// TIA Portal V15.1 export
// export: Created 2024-05-17T05:38:39.7334775Z, ExportSetting WithDefaults, DisplayName Totally Integrated Automation Portal, DisplayVersion V15.1 Update 5, DisplayName TIA Portal Openness, DisplayVersion V15.1 Update 5, DisplayName SINAMICS Startdrive Advanced, DisplayVersion V15.1, DisplayName G130, G150, S120, S150, SINAMICS MV, S210, DisplayVersion V15.1, DisplayName G110M, G120, G120C, G120D, G120P, DisplayVersion V15.1, DisplayName STEP 7 Professional, DisplayVersion V15.1 Update 5, DisplayName STEP 7 Safety, DisplayVersion V15.1, DisplayName WinCC Professional, DisplayVersion V15.1 Update 5, DisplayName SIMATIC Visualization Architect, DisplayVersion V15.1
FUNCTION_BLOCK "LGBJoyStick"   // FB6647, FBD
TITLE = LGBJoyStick
{ S7_Optimized_Access := 'TRUE' }
AUTHOR : VCC
FAMILY : Tooling
VERSION : 0.1
// ============================================================================
// This module works as a (virtual) joystick.
// The module can be used to force/block orders in a specific direction (lifts, cross conveyors, ...)
// ============================================================================
// stored: AutoNumber false, IsIECCheckEnabled true, IsRetainMemResEnabled false, MemoryReserve 100, SetENOAutomatically False, UDAEnableTagReadback false
   VAR_INPUT
      I_ExtBtnUp { ExternalAccessible := 'False'; ExternalVisible := 'False'; ExternalWritable := 'False'} : Bool;   // External Button Up
      I_ExtBtnRight { ExternalAccessible := 'False'; ExternalVisible := 'False'; ExternalWritable := 'False'} : Bool;   // External Button Right
      I_ExtBtnDown { ExternalAccessible := 'False'; ExternalVisible := 'False'; ExternalWritable := 'False'} : Bool;   // External Button Down
      I_ExtBtnLeft { ExternalAccessible := 'False'; ExternalVisible := 'False'; ExternalWritable := 'False'} : Bool;   // External Button Left
      I_OutOfUse { ExternalAccessible := 'False'; ExternalVisible := 'False'; ExternalWritable := 'False'} : Bool;   // Object out of use / Out of use
   END_VAR
   VAR_OUTPUT
      O_BtnMiddle { ExternalAccessible := 'False'; ExternalVisible := 'False'; ExternalWritable := 'False'} : Bool;   // Btn Middle Active
      O_BtnUp { ExternalAccessible := 'False'; ExternalVisible := 'False'; ExternalWritable := 'False'} : Bool;   // Btn Up Active
      O_BtnRight { ExternalAccessible := 'False'; ExternalVisible := 'False'; ExternalWritable := 'False'} : Bool;   // Btn Right Active
      O_BtnDown { ExternalAccessible := 'False'; ExternalVisible := 'False'; ExternalWritable := 'False'} : Bool;   // Btn Down Active
      O_BtnLeft { ExternalAccessible := 'False'; ExternalVisible := 'False'; ExternalWritable := 'False'} : Bool;   // Btn Left Active
      O_AnyBtnActive { ExternalAccessible := 'False'; ExternalVisible := 'False'; ExternalWritable := 'False'} : Bool;   // Any Button Active
      O_AlarmABCondition { ExternalAccessible := 'False'; ExternalVisible := 'False'; ExternalWritable := 'False'} : Bool;   // Alarm AB Condition
      O_AlarmA { ExternalAccessible := 'False'; ExternalVisible := 'False'; ExternalWritable := 'False'} : Bool;   // Alarm A
      O_AlarmB { ExternalAccessible := 'False'; ExternalVisible := 'False'; ExternalWritable := 'False'} : Bool;   // Alarm B
      O_AlarmC { ExternalAccessible := 'False'; ExternalVisible := 'False'; ExternalWritable := 'False'} : Bool;   // Alarm C
      O_AlarmD { ExternalAccessible := 'False'; ExternalVisible := 'False'; ExternalWritable := 'False'} : Bool;   // Alarm D
      H_AlarmDWord { ExternalAccessible := 'False'; ExternalVisible := 'False'; ExternalWritable := 'False'} : DWord;   // Alarm Word
   END_VAR
   VAR_IN_OUT
      H_HMI : "H_HMI";   // Icon Animation
      H_GBJoyStick : "H_GBJoyStick";   // Animation
      C_GBJoyStickConfig : "JoyStickConfig";   // Config
   END_VAR
   VAR
      AD_BtnMiddleActByHMI { ExternalAccessible := 'False'; ExternalVisible := 'False'; ExternalWritable := 'False'} : Bool;   // JoyStick - Button Middle is Active by HMI
      AD_BtnUpActByHMI { ExternalAccessible := 'False'; ExternalVisible := 'False'; ExternalWritable := 'False'} : Bool;   // JoyStick - Button Up is Active by HMI
      AD_BtnRightActByHMI { ExternalAccessible := 'False'; ExternalVisible := 'False'; ExternalWritable := 'False'} : Bool;   // JoyStick - Button Right is Active by HMI
      AD_BtnDownActByHMI { ExternalAccessible := 'False'; ExternalVisible := 'False'; ExternalWritable := 'False'} : Bool;   // JoyStick - Button Down is Active by HMI
      AD_BtnLeftActByHMI { ExternalAccessible := 'False'; ExternalVisible := 'False'; ExternalWritable := 'False'} : Bool;   // JoyStick - Button Left is Active by HMI
      AD_BtnUpActByExtCmd { ExternalAccessible := 'False'; ExternalVisible := 'False'; ExternalWritable := 'False'} : Bool;   // JoyStick - Button Up is Active by External command
      AD_BtnRightActByExtCmd { ExternalAccessible := 'False'; ExternalVisible := 'False'; ExternalWritable := 'False'} : Bool;   // JoyStick - Button Right is Active by External command
      AD_BtnDownActByExtCmd { ExternalAccessible := 'False'; ExternalVisible := 'False'; ExternalWritable := 'False'} : Bool;   // JoyStick - Button Down is Active by External command
      AD_BtnLeftActByExtCmd { ExternalAccessible := 'False'; ExternalVisible := 'False'; ExternalWritable := 'False'} : Bool;   // JoyStick - Button Left is Active by External command
      BtnHMICmd { ExternalAccessible := 'False'; ExternalVisible := 'False'; ExternalWritable := 'False'} : Struct   // HMI Commands
         BtnMiddle { ExternalAccessible := 'False'; ExternalVisible := 'False'; ExternalWritable := 'False'} : Bool;   // Btn Middle Selected
         BtnUp { ExternalAccessible := 'False'; ExternalVisible := 'False'; ExternalWritable := 'False'} : Bool;   // Btn Up Selected
         BtnRight { ExternalAccessible := 'False'; ExternalVisible := 'False'; ExternalWritable := 'False'} : Bool;   // Btn Right Selected
         BtnDown { ExternalAccessible := 'False'; ExternalVisible := 'False'; ExternalWritable := 'False'} : Bool;   // Btn Down Selected
         BtnLeft { ExternalAccessible := 'False'; ExternalVisible := 'False'; ExternalWritable := 'False'} : Bool;   // Btn Left Selected
      END_STRUCT;
      BtnResult { ExternalAccessible := 'False'; ExternalVisible := 'False'; ExternalWritable := 'False'} : Struct   // Buttons
         BtnMiddle { ExternalAccessible := 'False'; ExternalVisible := 'False'; ExternalWritable := 'False'} : Bool;   // Btn Middle Selected
         BtnUp { ExternalAccessible := 'False'; ExternalVisible := 'False'; ExternalWritable := 'False'} : Bool;   // Btn Up Selected
         BtnRight { ExternalAccessible := 'False'; ExternalVisible := 'False'; ExternalWritable := 'False'} : Bool;   // Btn Right Selected
         BtnDown { ExternalAccessible := 'False'; ExternalVisible := 'False'; ExternalWritable := 'False'} : Bool;   // Btn Down Selected
         BtnLeft { ExternalAccessible := 'False'; ExternalVisible := 'False'; ExternalWritable := 'False'} : Bool;   // Btn Left Selected
      END_STRUCT;
      Cmd { ExternalAccessible := 'False'; ExternalVisible := 'False'; ExternalWritable := 'False'} : Struct   // Commands
         Middle { ExternalAccessible := 'False'; ExternalVisible := 'False'; ExternalWritable := 'False'} : Bool;   // Middle Command
         BlockUp { ExternalAccessible := 'False'; ExternalVisible := 'False'; ExternalWritable := 'False'} : Bool;   // Block Up Command
         BlockRight { ExternalAccessible := 'False'; ExternalVisible := 'False'; ExternalWritable := 'False'} : Bool;   // Block Right Command
         BlockDown { ExternalAccessible := 'False'; ExternalVisible := 'False'; ExternalWritable := 'False'} : Bool;   // Block Down Command
         BlockLeft { ExternalAccessible := 'False'; ExternalVisible := 'False'; ExternalWritable := 'False'} : Bool;   // Block Left Command
         ForceUp { ExternalAccessible := 'False'; ExternalVisible := 'False'; ExternalWritable := 'False'} : Bool;   // Force Up Command
         ForceRight { ExternalAccessible := 'False'; ExternalVisible := 'False'; ExternalWritable := 'False'} : Bool;   // Force Right Command
         ForceDown { ExternalAccessible := 'False'; ExternalVisible := 'False'; ExternalWritable := 'False'} : Bool;   // Force Down Command
         ForceLeft { ExternalAccessible := 'False'; ExternalVisible := 'False'; ExternalWritable := 'False'} : Bool;   // Force Left Command
      END_STRUCT;
      Anim { ExternalAccessible := 'False'; ExternalVisible := 'False'; ExternalWritable := 'False'} : Struct   // HMI Animation
         HoldMiddleOff { ExternalAccessible := 'False'; ExternalVisible := 'False'; ExternalWritable := 'False'} : Bool;   // Anim Hold Middle Button Off
         HoldMiddleOn { ExternalAccessible := 'False'; ExternalVisible := 'False'; ExternalWritable := 'False'} : Bool;   // Anim Hold Middle Button On
         ForceUpOff { ExternalAccessible := 'False'; ExternalVisible := 'False'; ExternalWritable := 'False'} : Bool;   // Anim Force Up Button Off
         ForceUpOn { ExternalAccessible := 'False'; ExternalVisible := 'False'; ExternalWritable := 'False'} : Bool;   // Anim Force Up Button On
         BlockUpOff { ExternalAccessible := 'False'; ExternalVisible := 'False'; ExternalWritable := 'False'} : Bool;   // Anim Block Up Button Off
         BlockUpOn { ExternalAccessible := 'False'; ExternalVisible := 'False'; ExternalWritable := 'False'} : Bool;   // Anim Block Up Button On
         ForceRightOff { ExternalAccessible := 'False'; ExternalVisible := 'False'; ExternalWritable := 'False'} : Bool;   // Anim Force Right Button Off
         ForceRightOn { ExternalAccessible := 'False'; ExternalVisible := 'False'; ExternalWritable := 'False'} : Bool;   // Anim Force Right Button On
         BlockRightOff { ExternalAccessible := 'False'; ExternalVisible := 'False'; ExternalWritable := 'False'} : Bool;   // Anim Block Right Button Off
         BlockRightOn { ExternalAccessible := 'False'; ExternalVisible := 'False'; ExternalWritable := 'False'} : Bool;   // Anim Block Right Button On
         ForceDownOff { ExternalAccessible := 'False'; ExternalVisible := 'False'; ExternalWritable := 'False'} : Bool;   // Anim Force Down Button Off
         ForceDownOn { ExternalAccessible := 'False'; ExternalVisible := 'False'; ExternalWritable := 'False'} : Bool;   // Anim Force Down Button On
         BlockDownOff { ExternalAccessible := 'False'; ExternalVisible := 'False'; ExternalWritable := 'False'} : Bool;   // Anim Block Down Button Off
         BlockDownOn { ExternalAccessible := 'False'; ExternalVisible := 'False'; ExternalWritable := 'False'} : Bool;   // Anim Block Down Button On
         ForceLeftOff { ExternalAccessible := 'False'; ExternalVisible := 'False'; ExternalWritable := 'False'} : Bool;   // Anim Force Left Button Off
         ForceLeftOn { ExternalAccessible := 'False'; ExternalVisible := 'False'; ExternalWritable := 'False'} : Bool;   // Anim Force Left Button On
         BlockLeftOff { ExternalAccessible := 'False'; ExternalVisible := 'False'; ExternalWritable := 'False'} : Bool;   // Anim Block Left Button Off
         BlockLeftOn { ExternalAccessible := 'False'; ExternalVisible := 'False'; ExternalWritable := 'False'} : Bool;   // Anim Block Left Button On
      END_STRUCT;
      ExtBtnActive { ExternalAccessible := 'False'; ExternalVisible := 'False'; ExternalWritable := 'False'} : Bool;   // External Button Active
   END_VAR
   VAR RETAIN
      BtnMiddleAct { ExternalAccessible := 'False'; ExternalVisible := 'False'; ExternalWritable := 'False'} : Bool;   // Btn Middle Active memory
      BtnUpAct { ExternalAccessible := 'False'; ExternalVisible := 'False'; ExternalWritable := 'False'} : Bool;   // Btn Up Active memory
      BtnRightAct { ExternalAccessible := 'False'; ExternalVisible := 'False'; ExternalWritable := 'False'} : Bool;   // Btn Right Active memory
      BtnDownAct { ExternalAccessible := 'False'; ExternalVisible := 'False'; ExternalWritable := 'False'} : Bool;   // Btn Down Active memory
      BtnLeftAct { ExternalAccessible := 'False'; ExternalVisible := 'False'; ExternalWritable := 'False'} : Bool;   // Btn Left is Active memory
   END_VAR
   VAR
      AlarmA { ExternalAccessible := 'False'; ExternalVisible := 'False'; ExternalWritable := 'False'} : Bool;   // Alarm A
      AlarmB { ExternalAccessible := 'False'; ExternalVisible := 'False'; ExternalWritable := 'False'} : Bool;   // Alarm B
      AlarmC { ExternalAccessible := 'False'; ExternalVisible := 'False'; ExternalWritable := 'False'} : Bool;   // Alarm C
      AlarmD { ExternalAccessible := 'False'; ExternalVisible := 'False'; ExternalWritable := 'False'} : Bool;   // Alarm D
      Edge { ExternalAccessible := 'False'; ExternalVisible := 'False'; ExternalWritable := 'False'} : Array[0..10] of Bool;   // Edge
      ToggleMiddle { ExternalAccessible := 'False'; ExternalVisible := 'False'; ExternalWritable := 'False'} : "LToggle";   // FB
      ToggleUp { ExternalAccessible := 'False'; ExternalVisible := 'False'; ExternalWritable := 'False'} : "LToggle";   // FB
      ToggleRight { ExternalAccessible := 'False'; ExternalVisible := 'False'; ExternalWritable := 'False'} : "LToggle";   // FB
      ToggleDown { ExternalAccessible := 'False'; ExternalVisible := 'False'; ExternalWritable := 'False'} : "LToggle";   // FB
      ToggleLeft { ExternalAccessible := 'False'; ExternalVisible := 'False'; ExternalWritable := 'False'} : "LToggle";   // FB
   END_VAR
   VAR_TEMP   // added for the SCL form of the ladder/FBD networks
      _w1 : Bool;
      _w2 : Bool;
   END_VAR
BEGIN

REGION Network 1: **** 1 - Inputs **** Extract HMI Commands
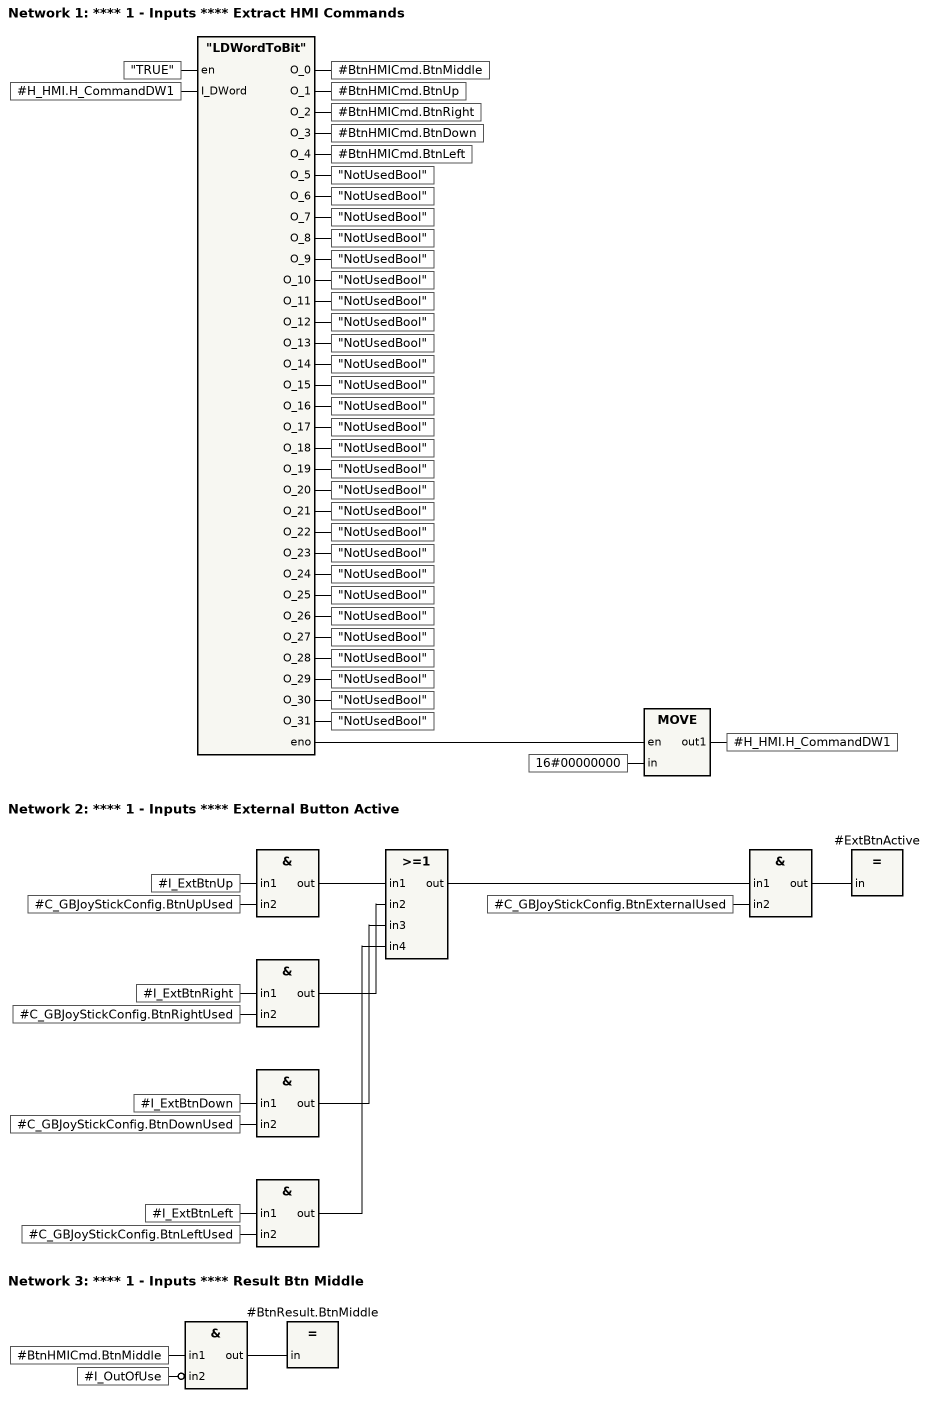
   "LDWordToBit"(EN := "TRUE",
                 I_DWord := #H_HMI.H_CommandDW1,
                 O_0 => #BtnHMICmd.BtnMiddle,
                 O_1 => #BtnHMICmd.BtnUp,
                 O_2 => #BtnHMICmd.BtnRight,
                 O_3 => #BtnHMICmd.BtnDown,
                 O_4 => #BtnHMICmd.BtnLeft,
                 O_5 => "NotUsedBool",
                 O_6 => "NotUsedBool",
                 O_7 => "NotUsedBool",
                 O_8 => "NotUsedBool",
                 O_9 => "NotUsedBool",
                 O_10 => "NotUsedBool",
                 O_11 => "NotUsedBool",
                 O_12 => "NotUsedBool",
                 O_13 => "NotUsedBool",
                 O_14 => "NotUsedBool",
                 O_15 => "NotUsedBool",
                 O_16 => "NotUsedBool",
                 O_17 => "NotUsedBool",
                 O_18 => "NotUsedBool",
                 O_19 => "NotUsedBool",
                 O_20 => "NotUsedBool",
                 O_21 => "NotUsedBool",
                 O_22 => "NotUsedBool",
                 O_23 => "NotUsedBool",
                 O_24 => "NotUsedBool",
                 O_25 => "NotUsedBool",
                 O_26 => "NotUsedBool",
                 O_27 => "NotUsedBool",
                 O_28 => "NotUsedBool",
                 O_29 => "NotUsedBool",
                 O_30 => "NotUsedBool",
                 O_31 => "NotUsedBool",
                 ENO => #_w1);
   IF #_w1 THEN #H_HMI.H_CommandDW1 := 16#00000000; END_IF;
END_REGION

REGION Network 2: **** 1 - Inputs **** External Button Active
   #ExtBtnActive := ((#I_ExtBtnUp AND #C_GBJoyStickConfig.BtnUpUsed) OR (#I_ExtBtnRight AND #C_GBJoyStickConfig.BtnRightUsed) OR (#I_ExtBtnDown AND #C_GBJoyStickConfig.BtnDownUsed) OR (#I_ExtBtnLeft AND #C_GBJoyStickConfig.BtnLeftUsed)) AND #C_GBJoyStickConfig.BtnExternalUsed;
END_REGION

REGION Network 3: **** 1 - Inputs **** Result Btn Middle
   #BtnResult.BtnMiddle := #BtnHMICmd.BtnMiddle AND NOT #I_OutOfUse;
END_REGION

REGION Network 4: **** 1 - Inputs **** Result Btn Up
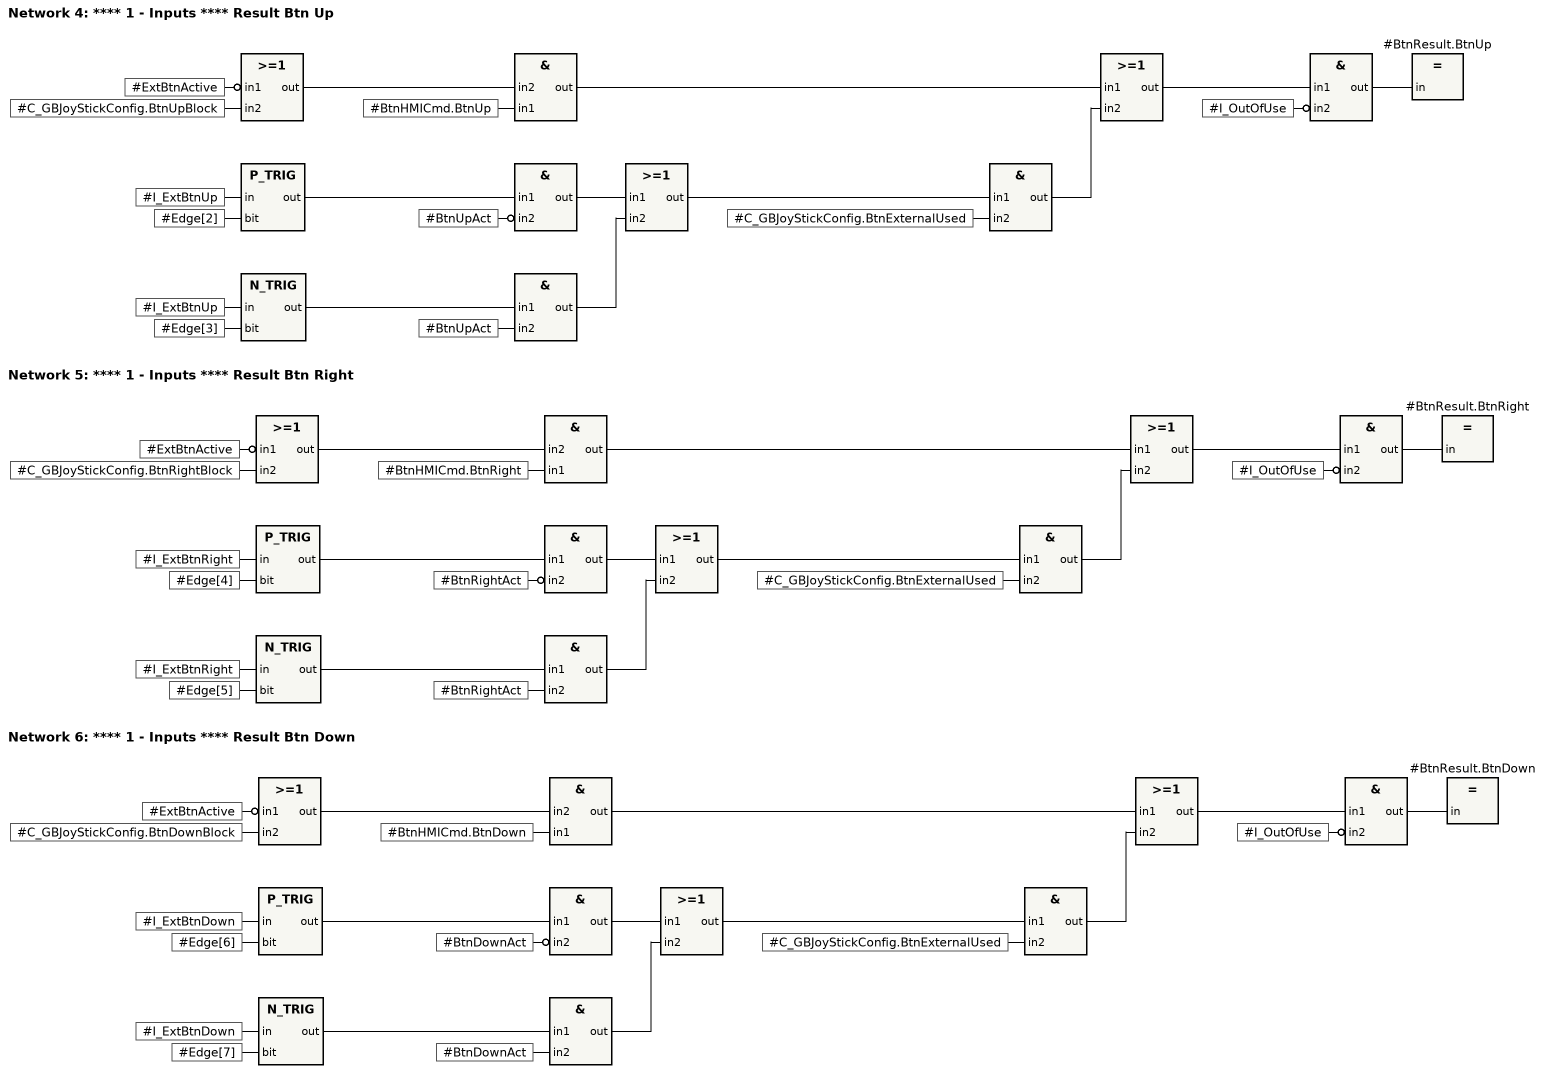
   #_w1 := #I_ExtBtnUp AND NOT #Edge[2];   // rising edge
   #Edge[2] := #I_ExtBtnUp;
   #_w2 := NOT #I_ExtBtnUp AND #Edge[3];   // falling edge
   #Edge[3] := #I_ExtBtnUp;
   #BtnResult.BtnUp := (((NOT #ExtBtnActive OR #C_GBJoyStickConfig.BtnUpBlock) AND #BtnHMICmd.BtnUp) OR (((#_w1 AND NOT #BtnUpAct) OR (#_w2 AND #BtnUpAct)) AND #C_GBJoyStickConfig.BtnExternalUsed)) AND NOT #I_OutOfUse;
END_REGION

REGION Network 5: **** 1 - Inputs **** Result Btn Right
   #_w1 := #I_ExtBtnRight AND NOT #Edge[4];   // rising edge
   #Edge[4] := #I_ExtBtnRight;
   #_w2 := NOT #I_ExtBtnRight AND #Edge[5];   // falling edge
   #Edge[5] := #I_ExtBtnRight;
   #BtnResult.BtnRight := (((NOT #ExtBtnActive OR #C_GBJoyStickConfig.BtnRightBlock) AND #BtnHMICmd.BtnRight) OR (((#_w1 AND NOT #BtnRightAct) OR (#_w2 AND #BtnRightAct)) AND #C_GBJoyStickConfig.BtnExternalUsed)) AND NOT #I_OutOfUse;
END_REGION

REGION Network 6: **** 1 - Inputs **** Result Btn Down
   #_w1 := #I_ExtBtnDown AND NOT #Edge[6];   // rising edge
   #Edge[6] := #I_ExtBtnDown;
   #_w2 := NOT #I_ExtBtnDown AND #Edge[7];   // falling edge
   #Edge[7] := #I_ExtBtnDown;
   #BtnResult.BtnDown := (((NOT #ExtBtnActive OR #C_GBJoyStickConfig.BtnDownBlock) AND #BtnHMICmd.BtnDown) OR (((#_w1 AND NOT #BtnDownAct) OR (#_w2 AND #BtnDownAct)) AND #C_GBJoyStickConfig.BtnExternalUsed)) AND NOT #I_OutOfUse;
END_REGION

REGION Network 7: **** 1 - Inputs **** Result Btn Left
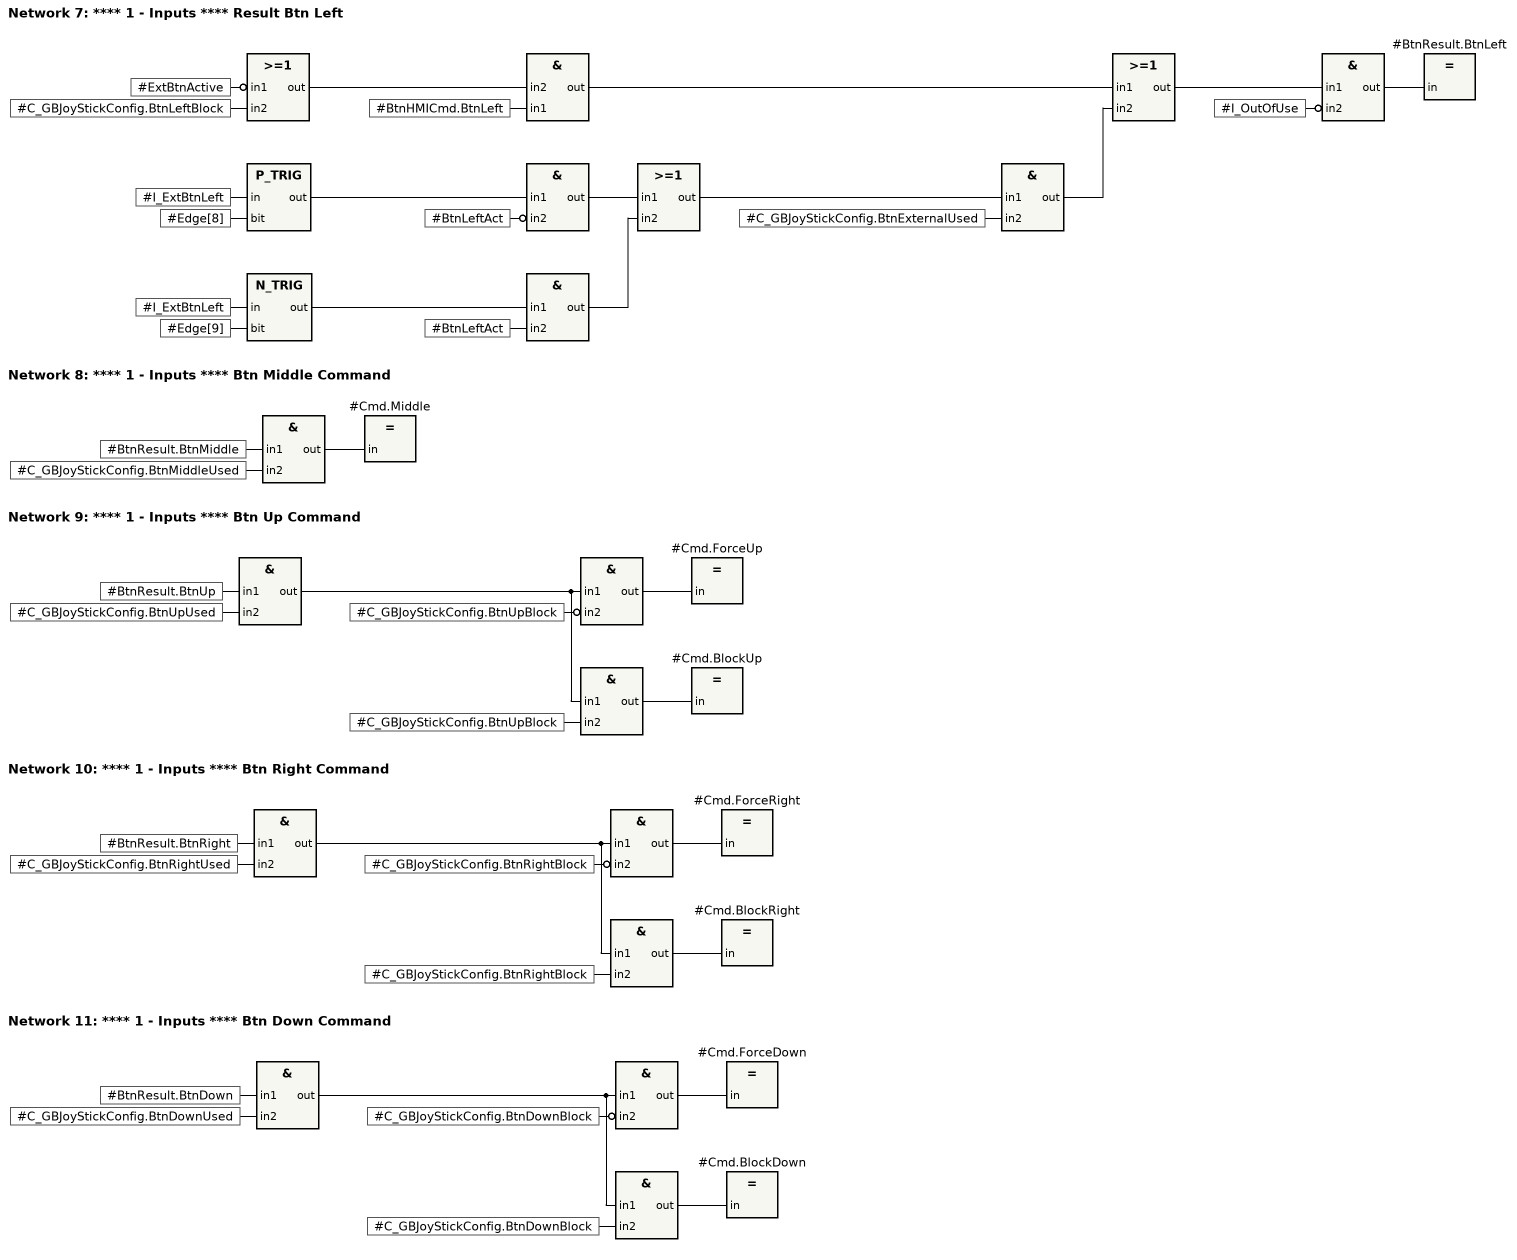
   #_w1 := #I_ExtBtnLeft AND NOT #Edge[8];   // rising edge
   #Edge[8] := #I_ExtBtnLeft;
   #_w2 := NOT #I_ExtBtnLeft AND #Edge[9];   // falling edge
   #Edge[9] := #I_ExtBtnLeft;
   #BtnResult.BtnLeft := (((NOT #ExtBtnActive OR #C_GBJoyStickConfig.BtnLeftBlock) AND #BtnHMICmd.BtnLeft) OR (((#_w1 AND NOT #BtnLeftAct) OR (#_w2 AND #BtnLeftAct)) AND #C_GBJoyStickConfig.BtnExternalUsed)) AND NOT #I_OutOfUse;
END_REGION

REGION Network 8: **** 1 - Inputs **** Btn Middle Command
   #Cmd.Middle := #BtnResult.BtnMiddle AND #C_GBJoyStickConfig.BtnMiddleUsed;
END_REGION

REGION Network 9: **** 1 - Inputs **** Btn Up Command
   #_w1 := #BtnResult.BtnUp AND #C_GBJoyStickConfig.BtnUpUsed;
   #Cmd.ForceUp := #_w1 AND NOT #C_GBJoyStickConfig.BtnUpBlock;
   #Cmd.BlockUp := #_w1 AND #C_GBJoyStickConfig.BtnUpBlock;
END_REGION

REGION Network 10: **** 1 - Inputs **** Btn Right Command
   #_w1 := #BtnResult.BtnRight AND #C_GBJoyStickConfig.BtnRightUsed;
   #Cmd.ForceRight := #_w1 AND NOT #C_GBJoyStickConfig.BtnRightBlock;
   #Cmd.BlockRight := #_w1 AND #C_GBJoyStickConfig.BtnRightBlock;
END_REGION

REGION Network 11: **** 1 - Inputs **** Btn Down Command
   #_w1 := #BtnResult.BtnDown AND #C_GBJoyStickConfig.BtnDownUsed;
   #Cmd.ForceDown := #_w1 AND NOT #C_GBJoyStickConfig.BtnDownBlock;
   #Cmd.BlockDown := #_w1 AND #C_GBJoyStickConfig.BtnDownBlock;
END_REGION

REGION Network 12: **** 1 - Inputs **** Btn Left Command
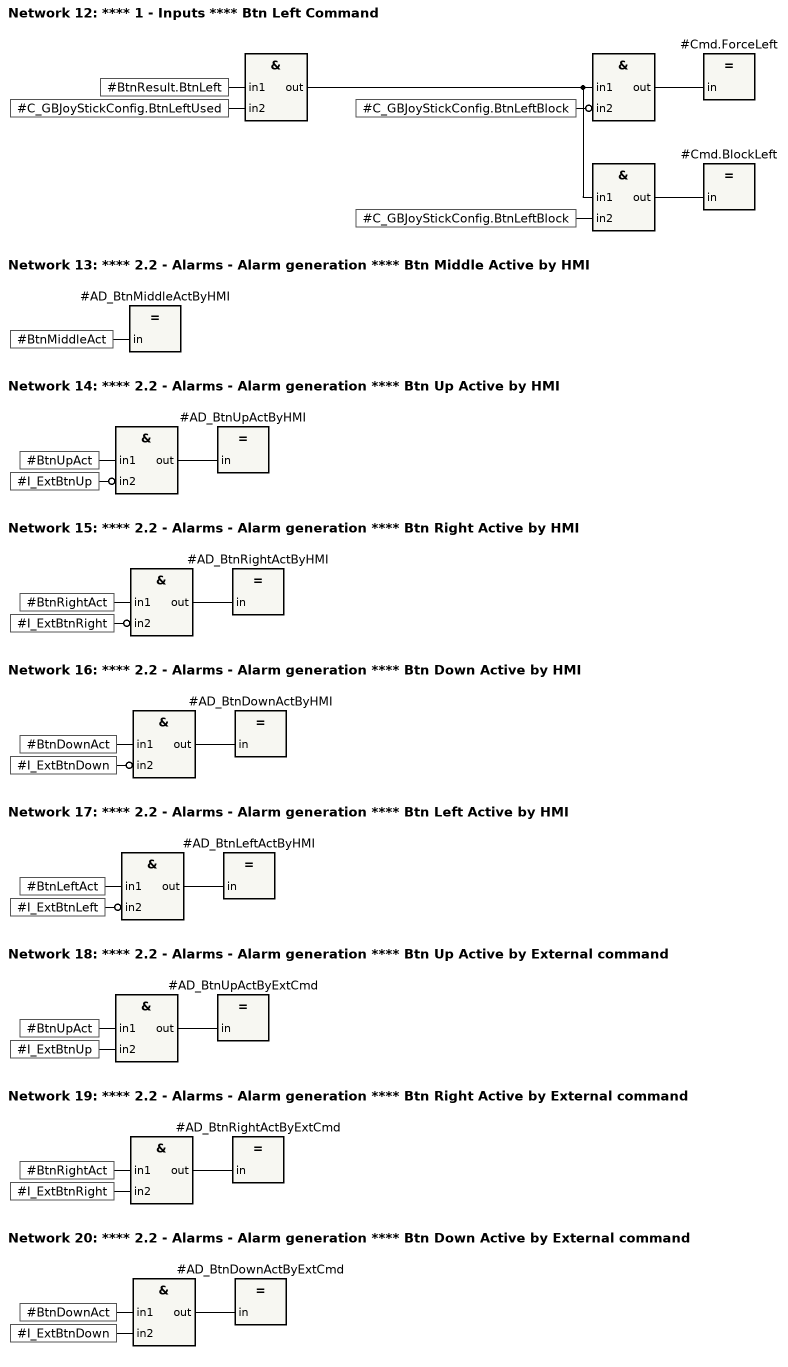
   #_w1 := #BtnResult.BtnLeft AND #C_GBJoyStickConfig.BtnLeftUsed;
   #Cmd.ForceLeft := #_w1 AND NOT #C_GBJoyStickConfig.BtnLeftBlock;
   #Cmd.BlockLeft := #_w1 AND #C_GBJoyStickConfig.BtnLeftBlock;
END_REGION

REGION Network 13: **** 2.2 - Alarms - Alarm generation **** Btn Middle Active by HMI
   #AD_BtnMiddleActByHMI := #BtnMiddleAct;
END_REGION

REGION Network 14: **** 2.2 - Alarms - Alarm generation **** Btn Up Active by HMI
   #AD_BtnUpActByHMI := #BtnUpAct AND NOT #I_ExtBtnUp;
END_REGION

REGION Network 15: **** 2.2 - Alarms - Alarm generation **** Btn Right Active by HMI
   #AD_BtnRightActByHMI := #BtnRightAct AND NOT #I_ExtBtnRight;
END_REGION

REGION Network 16: **** 2.2 - Alarms - Alarm generation **** Btn Down Active by HMI
   #AD_BtnDownActByHMI := #BtnDownAct AND NOT #I_ExtBtnDown;
END_REGION

REGION Network 17: **** 2.2 - Alarms - Alarm generation **** Btn Left Active by HMI
   #AD_BtnLeftActByHMI := #BtnLeftAct AND NOT #I_ExtBtnLeft;
END_REGION

REGION Network 18: **** 2.2 - Alarms - Alarm generation **** Btn Up Active by External command
   #AD_BtnUpActByExtCmd := #BtnUpAct AND #I_ExtBtnUp;
END_REGION

REGION Network 19: **** 2.2 - Alarms - Alarm generation **** Btn Right Active by External command
   #AD_BtnRightActByExtCmd := #BtnRightAct AND #I_ExtBtnRight;
END_REGION

REGION Network 20: **** 2.2 - Alarms - Alarm generation **** Btn Down Active by External command
   #AD_BtnDownActByExtCmd := #BtnDownAct AND #I_ExtBtnDown;
END_REGION

REGION Network 21: **** 2.2 - Alarms - Alarm generation **** Btn Left Active by External command
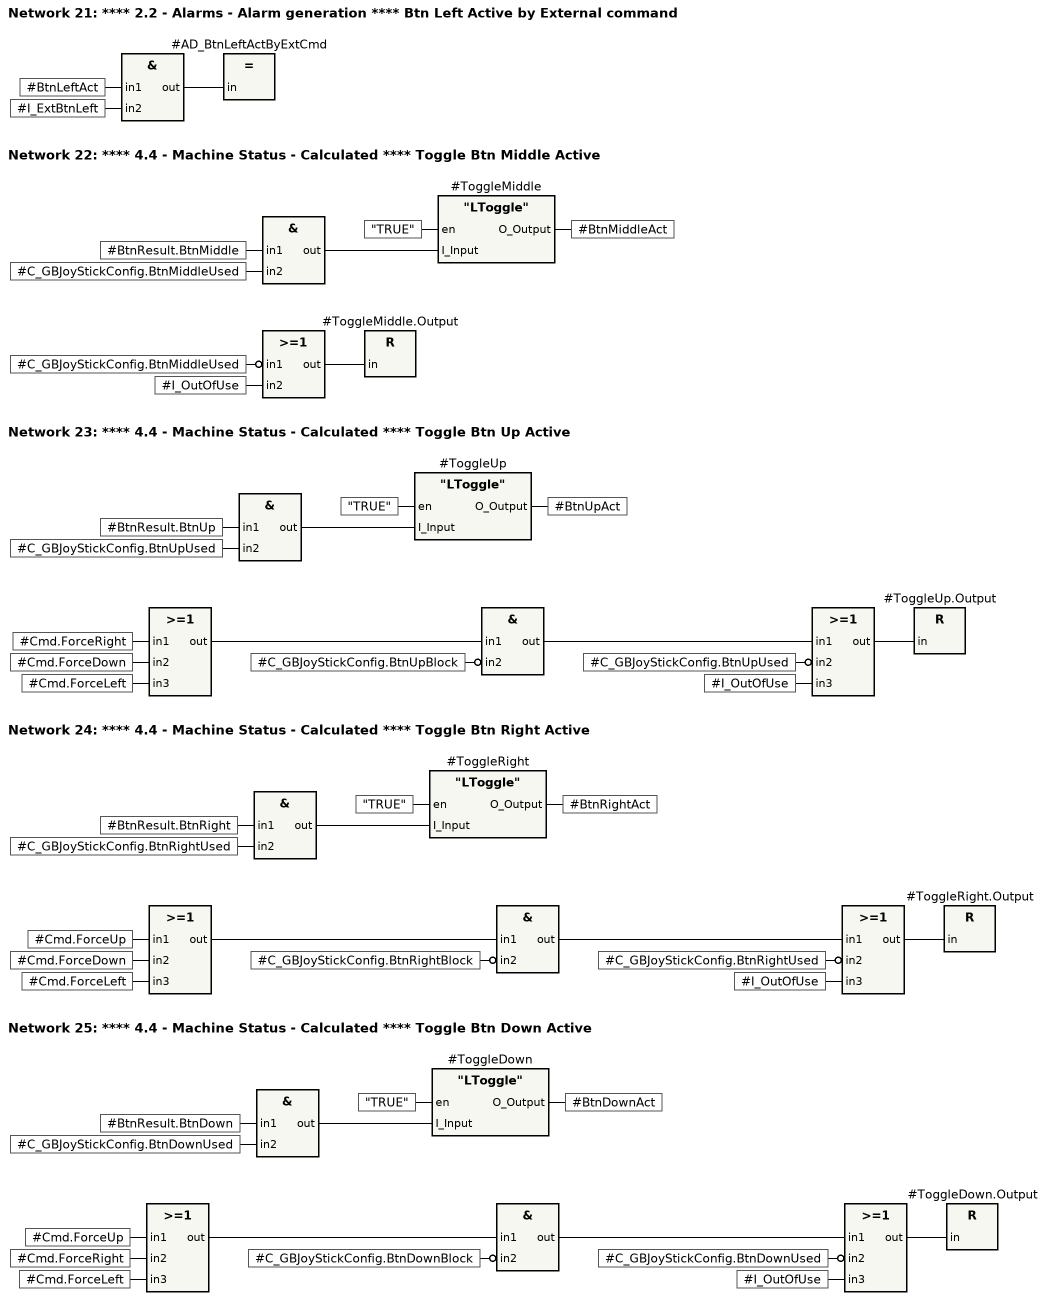
   #AD_BtnLeftActByExtCmd := #BtnLeftAct AND #I_ExtBtnLeft;
END_REGION

REGION Network 22: **** 4.4 - Machine Status - Calculated **** Toggle Btn Middle Active
   IF "TRUE" THEN
       #ToggleMiddle(I_Input := #BtnResult.BtnMiddle AND #C_GBJoyStickConfig.BtnMiddleUsed,   // "LToggle"
                     O_Output => #BtnMiddleAct);
   END_IF;
   IF NOT #C_GBJoyStickConfig.BtnMiddleUsed OR #I_OutOfUse THEN #ToggleMiddle.Output := FALSE; END_IF;
END_REGION

REGION Network 23: **** 4.4 - Machine Status - Calculated **** Toggle Btn Up Active
   IF "TRUE" THEN
       #ToggleUp(I_Input := #BtnResult.BtnUp AND #C_GBJoyStickConfig.BtnUpUsed, O_Output => #BtnUpAct);   // "LToggle"
   END_IF;
   IF ((#Cmd.ForceRight OR #Cmd.ForceDown OR #Cmd.ForceLeft) AND NOT #C_GBJoyStickConfig.BtnUpBlock) OR NOT #C_GBJoyStickConfig.BtnUpUsed OR #I_OutOfUse THEN
       #ToggleUp.Output := FALSE;
   END_IF;
END_REGION

REGION Network 24: **** 4.4 - Machine Status - Calculated **** Toggle Btn Right Active
   IF "TRUE" THEN
       #ToggleRight(I_Input := #BtnResult.BtnRight AND #C_GBJoyStickConfig.BtnRightUsed, O_Output => #BtnRightAct);   // "LToggle"
   END_IF;
   IF ((#Cmd.ForceUp OR #Cmd.ForceDown OR #Cmd.ForceLeft) AND NOT #C_GBJoyStickConfig.BtnRightBlock) OR NOT #C_GBJoyStickConfig.BtnRightUsed OR #I_OutOfUse THEN
       #ToggleRight.Output := FALSE;
   END_IF;
END_REGION

REGION Network 25: **** 4.4 - Machine Status - Calculated **** Toggle Btn Down Active
   IF "TRUE" THEN
       #ToggleDown(I_Input := #BtnResult.BtnDown AND #C_GBJoyStickConfig.BtnDownUsed, O_Output => #BtnDownAct);   // "LToggle"
   END_IF;
   IF ((#Cmd.ForceUp OR #Cmd.ForceRight OR #Cmd.ForceLeft) AND NOT #C_GBJoyStickConfig.BtnDownBlock) OR NOT #C_GBJoyStickConfig.BtnDownUsed OR #I_OutOfUse THEN
       #ToggleDown.Output := FALSE;
   END_IF;
END_REGION

REGION Network 26: **** 4.4 - Machine Status - Calculated **** Toggle Btn Left Active
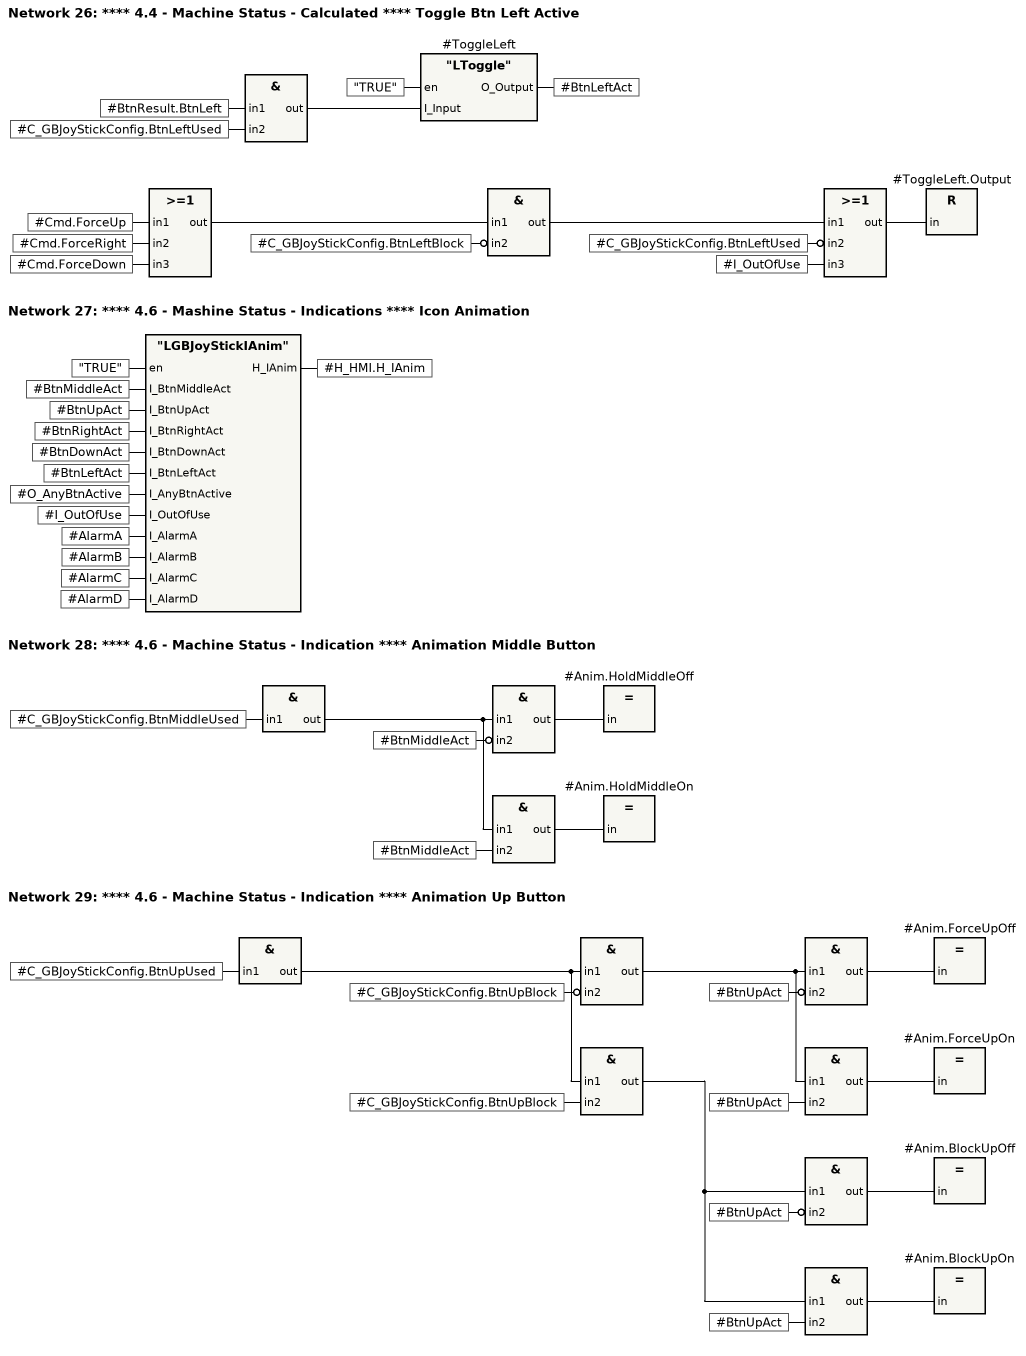
   IF "TRUE" THEN
       #ToggleLeft(I_Input := #BtnResult.BtnLeft AND #C_GBJoyStickConfig.BtnLeftUsed, O_Output => #BtnLeftAct);   // "LToggle"
   END_IF;
   IF ((#Cmd.ForceUp OR #Cmd.ForceRight OR #Cmd.ForceDown) AND NOT #C_GBJoyStickConfig.BtnLeftBlock) OR NOT #C_GBJoyStickConfig.BtnLeftUsed OR #I_OutOfUse THEN
       #ToggleLeft.Output := FALSE;
   END_IF;
END_REGION

REGION Network 27: **** 4.6 - Mashine Status - Indications **** Icon Animation
   // Icon Animation
   IF "TRUE" THEN
       "LGBJoyStickIAnim"(I_BtnMiddleAct := #BtnMiddleAct,
                          I_BtnUpAct := #BtnUpAct,
                          I_BtnRightAct := #BtnRightAct,
                          I_BtnDownAct := #BtnDownAct,
                          I_BtnLeftAct := #BtnLeftAct,
                          I_AnyBtnActive := #O_AnyBtnActive,
                          I_OutOfUse := #I_OutOfUse,
                          I_AlarmA := #AlarmA,
                          I_AlarmB := #AlarmB,
                          I_AlarmC := #AlarmC,
                          I_AlarmD := #AlarmD,
                          H_IAnim => #H_HMI.H_IAnim);
   END_IF;
END_REGION

REGION Network 28: **** 4.6 - Machine Status - Indication **** Animation Middle Button
   #Anim.HoldMiddleOff := #C_GBJoyStickConfig.BtnMiddleUsed AND NOT #BtnMiddleAct;
   #Anim.HoldMiddleOn := #C_GBJoyStickConfig.BtnMiddleUsed AND #BtnMiddleAct;
END_REGION

REGION Network 29: **** 4.6 - Machine Status - Indication **** Animation Up Button
   #_w1 := #C_GBJoyStickConfig.BtnUpUsed AND NOT #C_GBJoyStickConfig.BtnUpBlock;
   #Anim.ForceUpOff := #_w1 AND NOT #BtnUpAct;
   #Anim.ForceUpOn := #_w1 AND #BtnUpAct;
   #_w2 := #C_GBJoyStickConfig.BtnUpUsed AND #C_GBJoyStickConfig.BtnUpBlock;
   #Anim.BlockUpOff := #_w2 AND NOT #BtnUpAct;
   #Anim.BlockUpOn := #_w2 AND #BtnUpAct;
END_REGION

REGION Network 30: **** 4.6 - Machine Status - Indication **** Animation Right Button
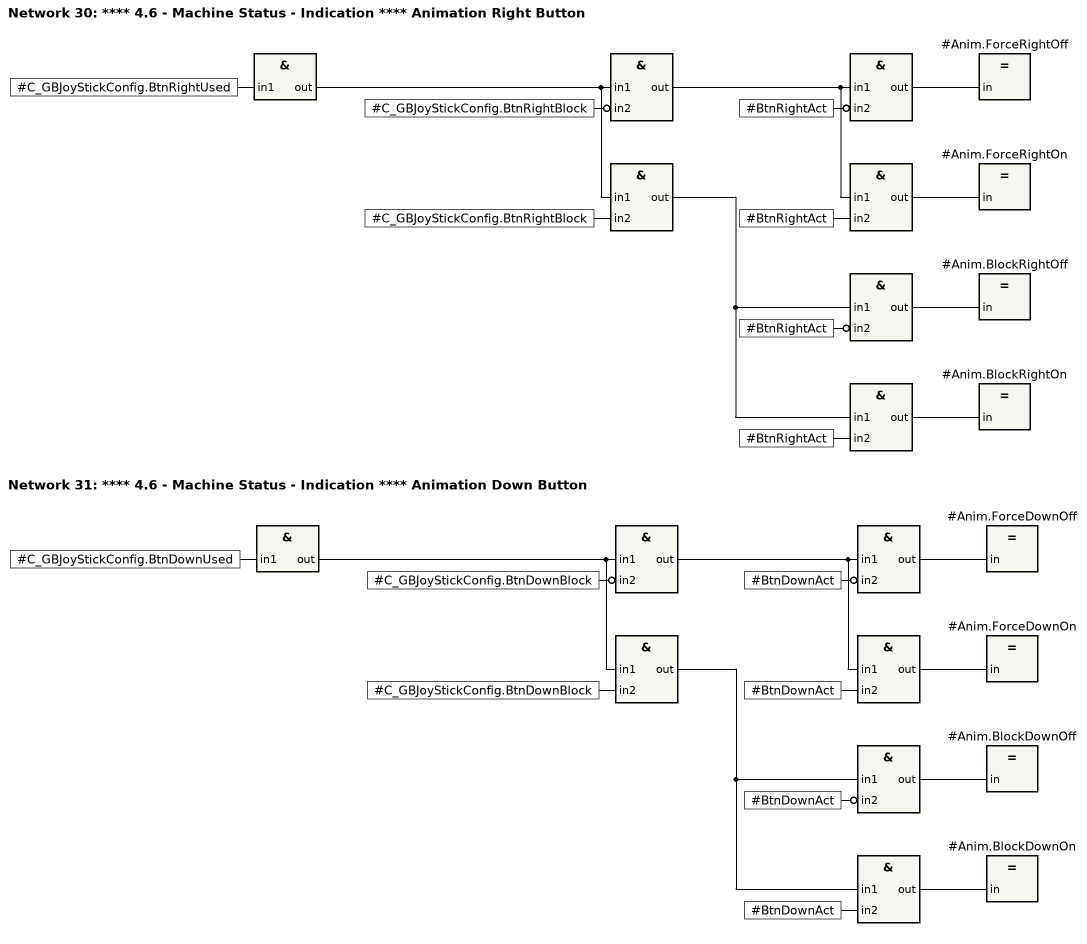
   #_w1 := #C_GBJoyStickConfig.BtnRightUsed AND NOT #C_GBJoyStickConfig.BtnRightBlock;
   #Anim.ForceRightOff := #_w1 AND NOT #BtnRightAct;
   #Anim.ForceRightOn := #_w1 AND #BtnRightAct;
   #_w2 := #C_GBJoyStickConfig.BtnRightUsed AND #C_GBJoyStickConfig.BtnRightBlock;
   #Anim.BlockRightOff := #_w2 AND NOT #BtnRightAct;
   #Anim.BlockRightOn := #_w2 AND #BtnRightAct;
END_REGION

REGION Network 31: **** 4.6 - Machine Status - Indication **** Animation Down Button
   #_w1 := #C_GBJoyStickConfig.BtnDownUsed AND NOT #C_GBJoyStickConfig.BtnDownBlock;
   #Anim.ForceDownOff := #_w1 AND NOT #BtnDownAct;
   #Anim.ForceDownOn := #_w1 AND #BtnDownAct;
   #_w2 := #C_GBJoyStickConfig.BtnDownUsed AND #C_GBJoyStickConfig.BtnDownBlock;
   #Anim.BlockDownOff := #_w2 AND NOT #BtnDownAct;
   #Anim.BlockDownOn := #_w2 AND #BtnDownAct;
END_REGION

REGION Network 32: **** 4.6 - Machine Status - Indication **** Animation Left Button
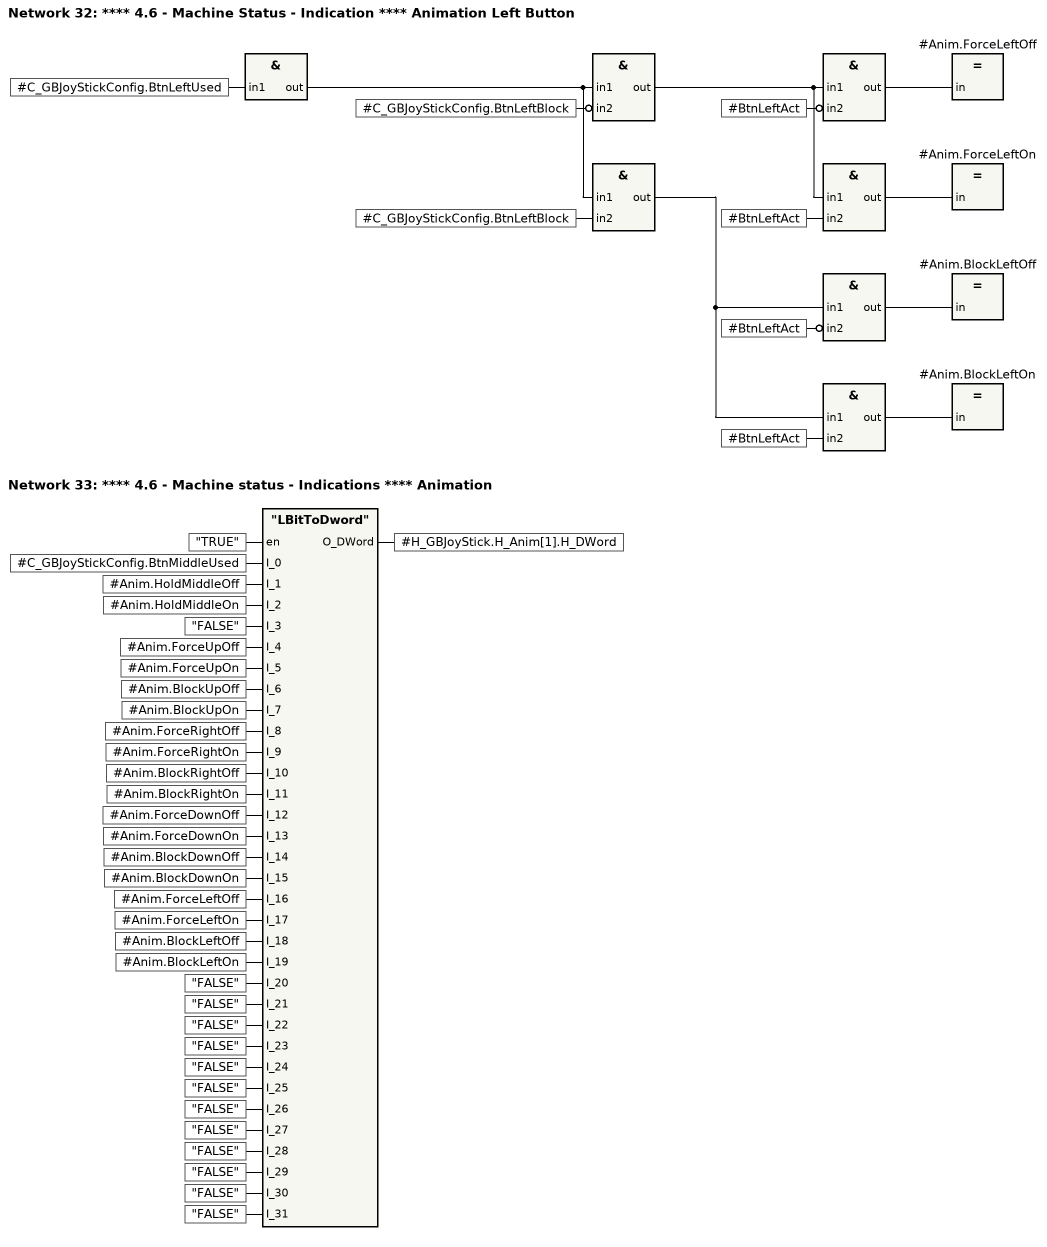
   #_w1 := #C_GBJoyStickConfig.BtnLeftUsed AND NOT #C_GBJoyStickConfig.BtnLeftBlock;
   #Anim.ForceLeftOff := #_w1 AND NOT #BtnLeftAct;
   #Anim.ForceLeftOn := #_w1 AND #BtnLeftAct;
   #_w2 := #C_GBJoyStickConfig.BtnLeftUsed AND #C_GBJoyStickConfig.BtnLeftBlock;
   #Anim.BlockLeftOff := #_w2 AND NOT #BtnLeftAct;
   #Anim.BlockLeftOn := #_w2 AND #BtnLeftAct;
END_REGION

REGION Network 33: **** 4.6 - Machine status - Indications **** Animation
   // Animation Word 1
   IF "TRUE" THEN
       "LBitToDword"(I_0 := #C_GBJoyStickConfig.BtnMiddleUsed,
                     I_1 := #Anim.HoldMiddleOff,
                     I_2 := #Anim.HoldMiddleOn,
                     I_3 := "FALSE",
                     I_4 := #Anim.ForceUpOff,
                     I_5 := #Anim.ForceUpOn,
                     I_6 := #Anim.BlockUpOff,
                     I_7 := #Anim.BlockUpOn,
                     I_8 := #Anim.ForceRightOff,
                     I_9 := #Anim.ForceRightOn,
                     I_10 := #Anim.BlockRightOff,
                     I_11 := #Anim.BlockRightOn,
                     I_12 := #Anim.ForceDownOff,
                     I_13 := #Anim.ForceDownOn,
                     I_14 := #Anim.BlockDownOff,
                     I_15 := #Anim.BlockDownOn,
                     I_16 := #Anim.ForceLeftOff,
                     I_17 := #Anim.ForceLeftOn,
                     I_18 := #Anim.BlockLeftOff,
                     I_19 := #Anim.BlockLeftOn,
                     I_20 := "FALSE",
                     I_21 := "FALSE",
                     I_22 := "FALSE",
                     I_23 := "FALSE",
                     I_24 := "FALSE",
                     I_25 := "FALSE",
                     I_26 := "FALSE",
                     I_27 := "FALSE",
                     I_28 := "FALSE",
                     I_29 := "FALSE",
                     I_30 := "FALSE",
                     I_31 := "FALSE",
                     O_DWord => #H_GBJoyStick.H_Anim[1].H_DWord);
   END_IF;
END_REGION

REGION Network 34: **** 4.6 - Machine status - Indications **** Animation
   // Animation Word 2
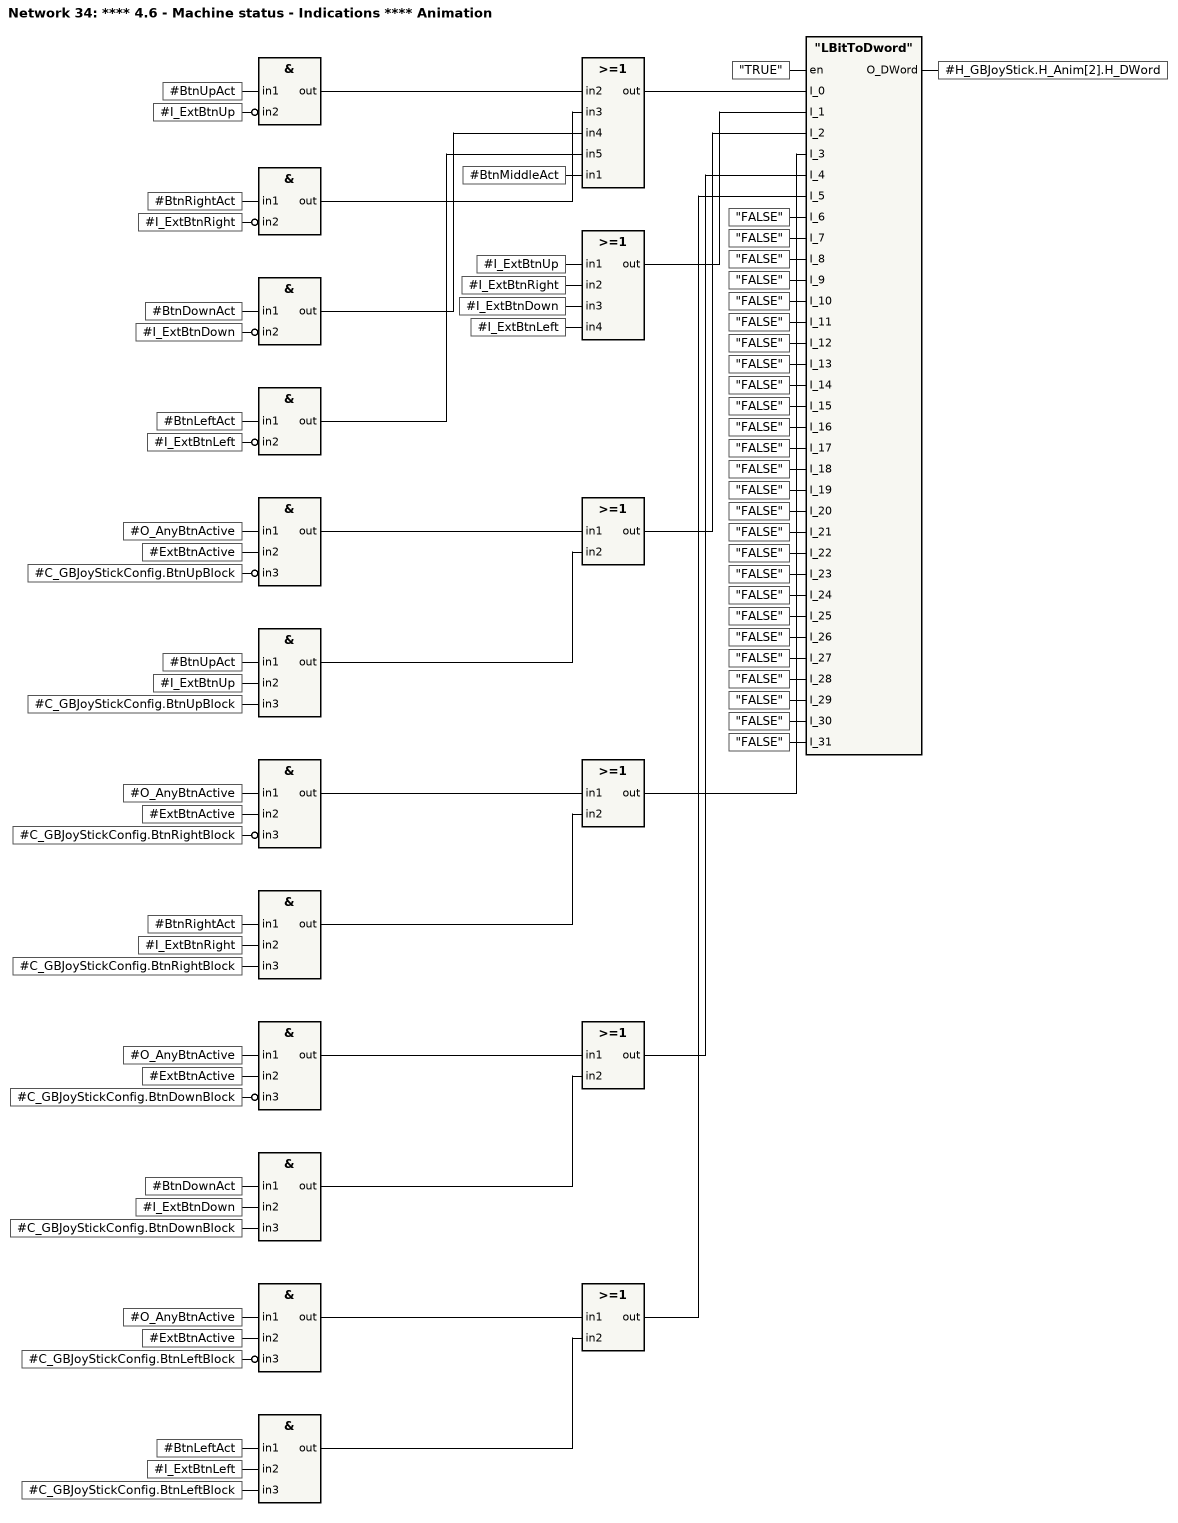
   IF "TRUE" THEN
       "LBitToDword"(I_0 := (#BtnUpAct AND NOT #I_ExtBtnUp) OR (#BtnRightAct AND NOT #I_ExtBtnRight) OR (#BtnDownAct AND NOT #I_ExtBtnDown) OR (#BtnLeftAct AND NOT #I_ExtBtnLeft) OR #BtnMiddleAct,
                     I_1 := #I_ExtBtnUp OR #I_ExtBtnRight OR #I_ExtBtnDown OR #I_ExtBtnLeft,
                     I_2 := (#O_AnyBtnActive AND #ExtBtnActive AND NOT #C_GBJoyStickConfig.BtnUpBlock) OR (#BtnUpAct AND #I_ExtBtnUp AND #C_GBJoyStickConfig.BtnUpBlock),
                     I_3 := (#O_AnyBtnActive AND #ExtBtnActive AND NOT #C_GBJoyStickConfig.BtnRightBlock) OR (#BtnRightAct AND #I_ExtBtnRight AND #C_GBJoyStickConfig.BtnRightBlock),
                     I_4 := (#O_AnyBtnActive AND #ExtBtnActive AND NOT #C_GBJoyStickConfig.BtnDownBlock) OR (#BtnDownAct AND #I_ExtBtnDown AND #C_GBJoyStickConfig.BtnDownBlock),
                     I_5 := (#O_AnyBtnActive AND #ExtBtnActive AND NOT #C_GBJoyStickConfig.BtnLeftBlock) OR (#BtnLeftAct AND #I_ExtBtnLeft AND #C_GBJoyStickConfig.BtnLeftBlock),
                     I_6 := "FALSE",
                     I_7 := "FALSE",
                     I_8 := "FALSE",
                     I_9 := "FALSE",
                     I_10 := "FALSE",
                     I_11 := "FALSE",
                     I_12 := "FALSE",
                     I_13 := "FALSE",
                     I_14 := "FALSE",
                     I_15 := "FALSE",
                     I_16 := "FALSE",
                     I_17 := "FALSE",
                     I_18 := "FALSE",
                     I_19 := "FALSE",
                     I_20 := "FALSE",
                     I_21 := "FALSE",
                     I_22 := "FALSE",
                     I_23 := "FALSE",
                     I_24 := "FALSE",
                     I_25 := "FALSE",
                     I_26 := "FALSE",
                     I_27 := "FALSE",
                     I_28 := "FALSE",
                     I_29 := "FALSE",
                     I_30 := "FALSE",
                     I_31 := "FALSE",
                     O_DWord => #H_GBJoyStick.H_Anim[2].H_DWord);
   END_IF;
END_REGION

REGION Network 35: **** 4.6 - Machine status - Indications **** Animation Text
   // Animation Text
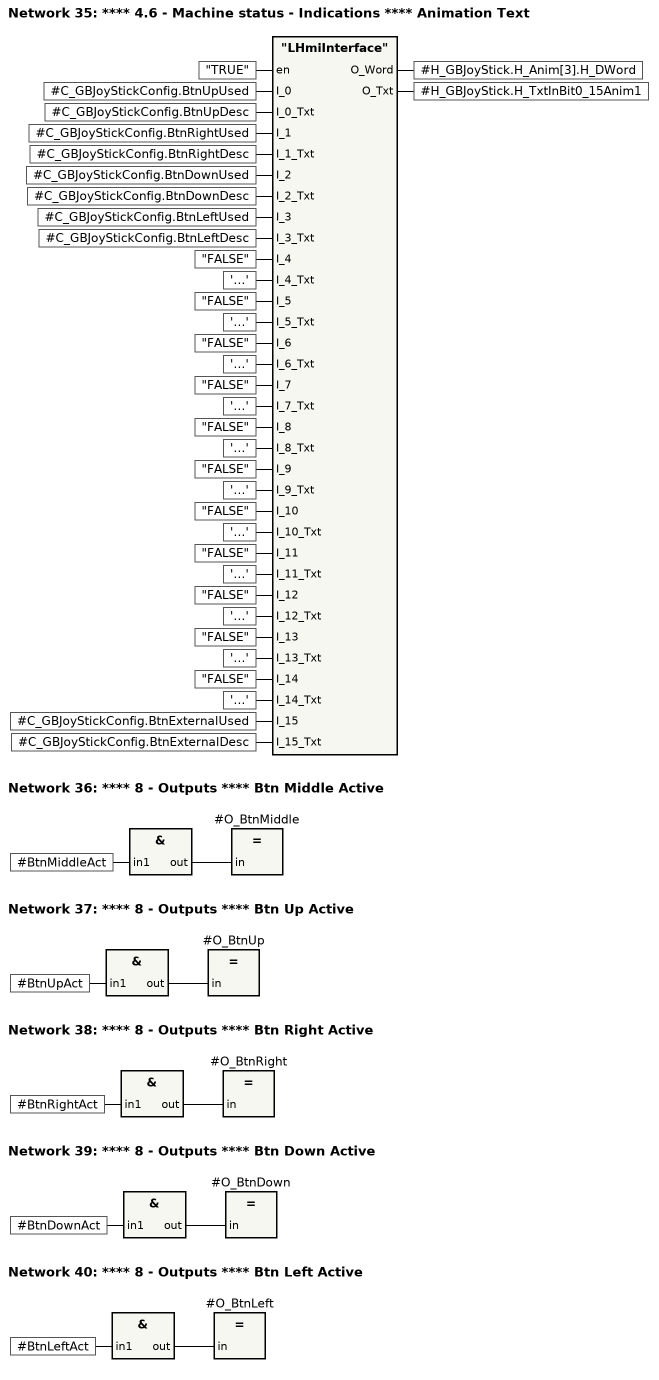
   IF "TRUE" THEN
       "LHmiInterface"(I_0 := #C_GBJoyStickConfig.BtnUpUsed,
                       I_0_Txt := #C_GBJoyStickConfig.BtnUpDesc,
                       I_1 := #C_GBJoyStickConfig.BtnRightUsed,
                       I_1_Txt := #C_GBJoyStickConfig.BtnRightDesc,
                       I_2 := #C_GBJoyStickConfig.BtnDownUsed,
                       I_2_Txt := #C_GBJoyStickConfig.BtnDownDesc,
                       I_3 := #C_GBJoyStickConfig.BtnLeftUsed,
                       I_3_Txt := #C_GBJoyStickConfig.BtnLeftDesc,
                       I_4 := "FALSE",
                       I_4_Txt := '...',
                       I_5 := "FALSE",
                       I_5_Txt := '...',
                       I_6 := "FALSE",
                       I_6_Txt := '...',
                       I_7 := "FALSE",
                       I_7_Txt := '...',
                       I_8 := "FALSE",
                       I_8_Txt := '...',
                       I_9 := "FALSE",
                       I_9_Txt := '...',
                       I_10 := "FALSE",
                       I_10_Txt := '...',
                       I_11 := "FALSE",
                       I_11_Txt := '...',
                       I_12 := "FALSE",
                       I_12_Txt := '...',
                       I_13 := "FALSE",
                       I_13_Txt := '...',
                       I_14 := "FALSE",
                       I_14_Txt := '...',
                       I_15 := #C_GBJoyStickConfig.BtnExternalUsed,
                       I_15_Txt := #C_GBJoyStickConfig.BtnExternalDesc,
                       O_Word => #H_GBJoyStick.H_Anim[3].H_DWord,
                       O_Txt => #H_GBJoyStick.H_TxtInBit0_15Anim1);
   END_IF;
END_REGION

REGION Network 36: **** 8 - Outputs **** Btn Middle Active
   #O_BtnMiddle := #BtnMiddleAct;
END_REGION

REGION Network 37: **** 8 - Outputs **** Btn Up Active
   #O_BtnUp := #BtnUpAct;
END_REGION

REGION Network 38: **** 8 - Outputs **** Btn Right Active
   #O_BtnRight := #BtnRightAct;
END_REGION

REGION Network 39: **** 8 - Outputs **** Btn Down Active
   #O_BtnDown := #BtnDownAct;
END_REGION

REGION Network 40: **** 8 - Outputs **** Btn Left Active
   #O_BtnLeft := #BtnLeftAct;
END_REGION

REGION Network 41: **** 8 - Outputs **** Any Btn Active
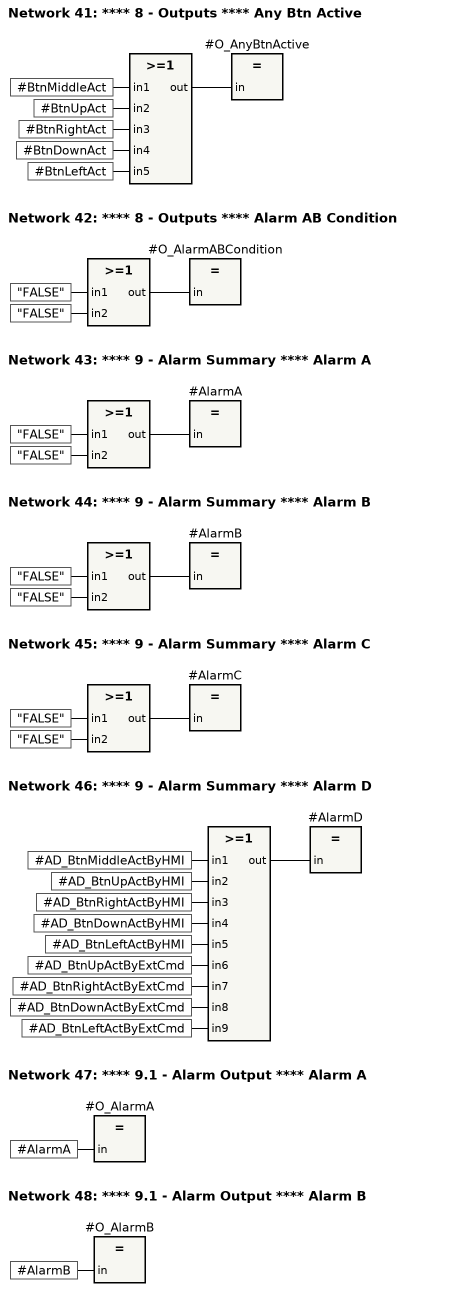
   #O_AnyBtnActive := #BtnMiddleAct OR #BtnUpAct OR #BtnRightAct OR #BtnDownAct OR #BtnLeftAct;
END_REGION

REGION Network 42: **** 8 - Outputs **** Alarm AB Condition
   // Alarm AB Condition
   #O_AlarmABCondition := "FALSE" OR "FALSE";
END_REGION

REGION Network 43: **** 9 - Alarm Summary **** Alarm A
   // Alarm A
   #AlarmA := "FALSE" OR "FALSE";
END_REGION

REGION Network 44: **** 9 - Alarm Summary **** Alarm B
   // Alarm B
   #AlarmB := "FALSE" OR "FALSE";
END_REGION

REGION Network 45: **** 9 - Alarm Summary **** Alarm C
   // Alarm C
   #AlarmC := "FALSE" OR "FALSE";
END_REGION

REGION Network 46: **** 9 - Alarm Summary **** Alarm D
   // Alarm D
   #AlarmD := #AD_BtnMiddleActByHMI OR #AD_BtnUpActByHMI OR #AD_BtnRightActByHMI OR #AD_BtnDownActByHMI OR #AD_BtnLeftActByHMI OR #AD_BtnUpActByExtCmd OR #AD_BtnRightActByExtCmd OR #AD_BtnDownActByExtCmd OR #AD_BtnLeftActByExtCmd;
END_REGION

REGION Network 47: **** 9.1 - Alarm Output **** Alarm A
   // Alarm A
   #O_AlarmA := #AlarmA;
END_REGION

REGION Network 48: **** 9.1 - Alarm Output **** Alarm B
   // Alarm B
   #O_AlarmB := #AlarmB;
END_REGION

REGION Network 49: **** 9.1 - Alarm Output **** Alarm C
   // Alarm C
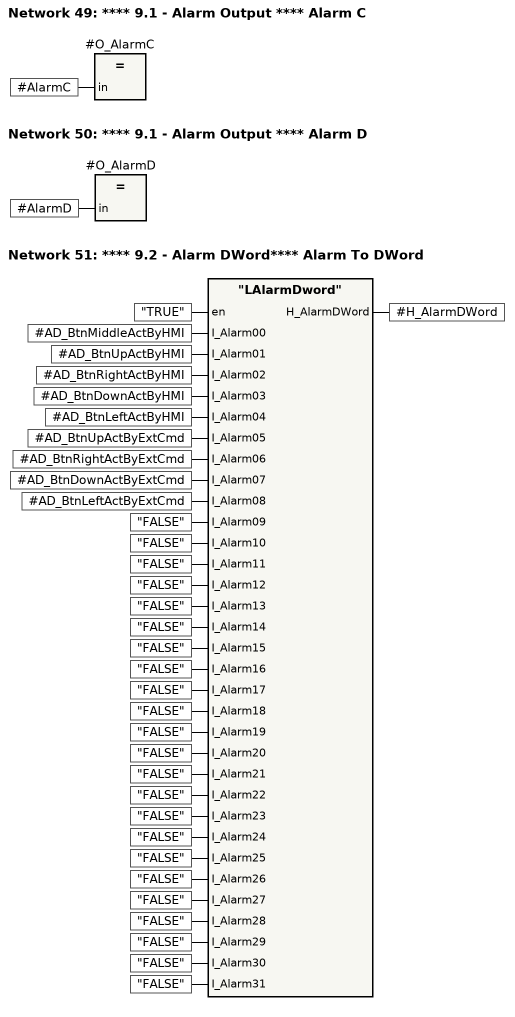
   #O_AlarmC := #AlarmC;
END_REGION

REGION Network 50: **** 9.1 - Alarm Output **** Alarm D
   // Alarm D
   #O_AlarmD := #AlarmD;
END_REGION

REGION Network 51: **** 9.2 - Alarm DWord**** Alarm To DWord
   // Alarm To DWord
   IF "TRUE" THEN
       "LAlarmDword"(I_Alarm00 := #AD_BtnMiddleActByHMI,
                     I_Alarm01 := #AD_BtnUpActByHMI,
                     I_Alarm02 := #AD_BtnRightActByHMI,
                     I_Alarm03 := #AD_BtnDownActByHMI,
                     I_Alarm04 := #AD_BtnLeftActByHMI,
                     I_Alarm05 := #AD_BtnUpActByExtCmd,
                     I_Alarm06 := #AD_BtnRightActByExtCmd,
                     I_Alarm07 := #AD_BtnDownActByExtCmd,
                     I_Alarm08 := #AD_BtnLeftActByExtCmd,
                     I_Alarm09 := "FALSE",
                     I_Alarm10 := "FALSE",
                     I_Alarm11 := "FALSE",
                     I_Alarm12 := "FALSE",
                     I_Alarm13 := "FALSE",
                     I_Alarm14 := "FALSE",
                     I_Alarm15 := "FALSE",
                     I_Alarm16 := "FALSE",
                     I_Alarm17 := "FALSE",
                     I_Alarm18 := "FALSE",
                     I_Alarm19 := "FALSE",
                     I_Alarm20 := "FALSE",
                     I_Alarm21 := "FALSE",
                     I_Alarm22 := "FALSE",
                     I_Alarm23 := "FALSE",
                     I_Alarm24 := "FALSE",
                     I_Alarm25 := "FALSE",
                     I_Alarm26 := "FALSE",
                     I_Alarm27 := "FALSE",
                     I_Alarm28 := "FALSE",
                     I_Alarm29 := "FALSE",
                     I_Alarm30 := "FALSE",
                     I_Alarm31 := "FALSE",
                     H_AlarmDWord => #H_AlarmDWord);
   END_IF;
END_REGION
END_FUNCTION_BLOCK
